FUNCTION_BLOCK ClientDataExchanger
VAR_INPUT
END_VAR
VAR_OUTPUT
END_VAR
VAR
	//TODO: Finish https://infosys.beckhoff.com/english.php?content=../content/1033/tf6310_tc3_tcpip/84203915.html&id=
	//Note: Needed? Wouldn't it be better to just have a .Send and .Receive methods?
	m_socketHandle : T_HSOCKET;
	m_messageToServer : T_MaxString;	

END_VAR

END_FUNCTION_BLOCK

(* stored: Version 1.1.0.1, ProductVersion 3.1.4024.12
   POU ClientDataExchanger: Id {4c6b4c11-d030-47d4-aaf8-df7c8a8bffa3}, SpecialFunc None *)
